(* PLC project Generated.project, CODESYS CODESYS V3.5 SP19 Patch 1 *)
(* stored: creationDateTime 2026-09-06T13:00:42.471378, modificationDateTime 2026-09-06T13:00:42.471378 *)

(* ======================================================================= ⚙️ ST_fbEncoder_Cfg — Réglages technologiques publics de FB_Encoder ─────────────────────────────────────────────────────────────────────── 🎯 Rôle : porter le mode de confirmation preset commun aux codeurs. 🔒 Ownership : GVL_IHM.Commun.EncoderCfg ↔ GVL_PERSISTENT._EncoderCfgPersist. 📄 Doc : DOC/AF/AF_Partie-09_Fonction_Encoder_v2.4.md ======================================================================= *)
TYPE ST_fbEncoder_Cfg : STRUCT
  PresetConfirmMode : E_PresetConfirmMode := E_PresetConfirmMode.READBACK_ONLY;  (* Mode de confirmation preset, défaut relecture *)
  Initialized : BOOL := FALSE;  (* 🚦 TRUE après restauration du pont persistant *)
END_STRUCT;
END_TYPE

(* values of E_PresetConfirmMode: READBACK_ONLY: Confirmation par relecture de position; READBACK_AND_STATUSBIT: Relecture et bit d'état matériel; STATUSBIT_ONLY: Bit d'état matériel uniquement *)

{attribute 'qualified_only'}
{attribute 'strict'}
TYPE E_PresetConfirmMode : (READBACK_ONLY := 0, READBACK_AND_STATUSBIT := 1, STATUSBIT_ONLY := 2);
END_TYPE

(* ======================================================================= 💾 FB_CfgPersistBridge_fbEncoder_Cfg — Pont persistance pour ST_fbEncoder_Cfg ─────────────────────────────────────────────────────────────────────── 🎯 Rôle : restauration et synchronisation bidirectionnelle IHM / Persist. 💾 Persistance : transfert GVL_PERSISTENT <-> GVL_IHM sur Initialized. 📄 Doc : DOC/AF/AF_Partie-09_Fonction_Encoder_v2.4.md ======================================================================= *)
FUNCTION_BLOCK FB_CfgPersistBridge_fbEncoder_Cfg
  VAR_OUTPUT
    JustRestored : BOOL;  (* === ETATS RESTAURATION === <-- [STAT] Vrai sur le cycle de restauration initiale *)
  END_VAR
  VAR_IN_OUT
    Hmi : ST_fbEncoder_Cfg;  (* === BUS CONFIGURATION ET PERSISTANCE === <-> [BUS] Structure de configuration IHM commune *)
    Persist : ST_fbEncoder_Cfg;  (* <-> [BUS] Structure de configuration persistante *)
  END_VAR

            

JustRestored := FALSE;
IF NOT Hmi.Initialized THEN
    Hmi := Persist;
    Hmi.Initialized := TRUE;
    JustRestored := TRUE;
ELSE
    Persist := Hmi;
END_IF;

          
END_FUNCTION_BLOCK
